// TIA Portal V20 export
// export: Created 2025-12-01T14:57:43.22394Z, ExportSetting None, DisplayName Totally Integrated Automation Portal, DisplayVersion V20 Update 3, DisplayName TIA Portal Openness, DisplayVersion V20 Update 3, DisplayName TIA Portal Version Control Interface, DisplayVersion V20 Update 3, DisplayName STEP 7 Professional, DisplayVersion V20 Update 3, DisplayName STEP 7 Safety, DisplayVersion V20 Update 2, DisplayName WinCC Basic/Comfort/Advanced, DisplayVersion V20 Update 3, DisplayName WinCC Professional, DisplayVersion V20 Update 3, DisplayName WinCC Unified, DisplayVersion V20 Update 3
DATA_BLOCK "FB955_Leer_Ips_Gateways_DB"   // DB955
// stored: AutoNumber false, InstanceOfName FB955_Leer_Ips_Gateways, InstanceOfType FB
"FB955_Leer_Ips_Gateways"
   // VAR
   //    Gateway { S7_SetPoint := 'True'} : Array[1..16] of "LPNDR_ReadGlobalInfo";
   //    lee { S7_SetPoint := 'True'} : Array[1..16] of Bool;
   // END_VAR
BEGIN
END_DATA_BLOCK
